// TwinCAT 3 PLC project CSVExample
// ProgramVersion: 3.1.0.8
// libraries:
//   Tc2_Standard, * (Beckhoff Automation GmbH)
//   Tc2_System, * (Beckhoff Automation GmbH)
//   Tc2_Utilities, * (Beckhoff Automation GmbH)
//   Tc3_Interfaces, * (Beckhoff Automation GmbH)
//   Tc3_Module, * (Beckhoff Automation GmbH)
// project tree:
//   DUTs/ ST_CSV_Record.TcDUT (not stored)
//   GVLs/ GVL.TcGVL
//   POUs/CSV read_write in binary mode/ P_BinaryModeRead.TcPOU (not stored), P_BinaryModeWrite.TcPOU (not stored)
//   POUs/CSV read_write in text mode/ P_TextModeRead.TcPOU (not stored), P_TextModeWrite.TcPOU (not stored)
//   POUs/ MAIN.TcPOU, P_ArgToConvExample.TcPOU (not stored), P_StringToConvExample.TcPOU (not stored)
//   / PlcTask.TcTTO (not stored)

// ---- GVLs/GVL.TcGVL
VAR_GLOBAL CONSTANT
	MAX_CSV_ROWS 			: UDINT := 100;
	MAX_CSV_COLUMNS 		: UDINT := 5;
	MAX_CSV_FIELD_LENGTH	: UDINT := 100;
END_VAR

// ---- POUs/MAIN.TcPOU
PROGRAM MAIN
VAR
(*	In USA/UK the CSV field separator is a comma.
	In Germany and some other European countries the CSV field separator is a semicolon. *)
	bChangeSeparatorToComma	: BOOL := FALSE;
END_VAR

IF bChangeSeparatorToComma THEN
	DEFAULT_CSV_FIELD_SEP := 16#2C;(* Comma ASCII code *)
ELSE
	DEFAULT_CSV_FIELD_SEP := 16#3B;(* Semicolon ASCII code *)
END_IF

P_TextModeRead();(* This sample program opens and reads CSV file in text mode *)

P_TextModeWrite();(* This sample program opens and writes CSV file in text mode *)

P_BinaryModeRead();(* This sample program opens and reads CSV file in binary mode *)

P_BinaryModeWrite();(* This sample program opens and writes CSV file in binary mode *)

P_ArgToConvExample();(* This sample program shows the usage of the ARG_TO_CSVFIELD and CSVFILED_TO_ARG conversion functions *)

P_StringToConvExample();(* This sample program shows the usage of the STRING_TO_CSVFIELD and CSVFIELD_TO_STRING conversion functions *)

END_PROGRAM
